FUNCTION_BLOCK CurtainControl EXTENDS Curtain
VAR
	OpenCmd AT%I* : BOOL;
	CloseCmd AT%I* : BOOL;
	
	App_OpenCmd: BOOL;
	App_CloseCmd: BOOL;

END_VAR


	IF (OpenCmd OR App_OpenCmd) AND ((NOT CloseCmd) OR (NOT App_CloseCmd)) THEN
		Open(IN	:=	TRUE);
	ELSE
		Open(IN	:=	FALSE);
	END_IF

	IF (CloseCmd OR App_CloseCmd) AND ((NOT OpenCmd) OR (NOT App_OpenCmd)) THEN
		Close(IN	:=	TRUE);
	ELSE
		Close(IN	:=	FALSE);
	END_IF

	IF (OpenCmd AND CloseCmd) OR (App_OpenCmd AND App_CloseCmd) THEN
		Open(IN	:=	FALSE);
		Close(IN	:=	FALSE);
	END_IF

END_FUNCTION_BLOCK

(* stored: Version 1.1.0.1, ProductVersion 3.1.4024.13
   POU CurtainControl: Id {4b2829aa-3204-4a26-9487-5be3e74830bb}, SpecialFunc None *)
